{attribute 'linkalways'} 
{attribute 'no_explicit_call' := 'This FB is a CLASS and must be accessed using methods or properties'}
{attribute 'enable_dynamic_creation'}
FUNCTION_BLOCK _ETcVnColorMapSize EXTENDS EnumDatatypeBase
VAR
	localData : ETcVnColorMapSize;
	activeData : REFERENCE TO ETcVnColorMapSize;
	enumBaseDatatype : _UDINT(localData);
END_VAR

METHOD PRIVATE AddLocalEnumeration
VAR_INPUT
	Enumeration : T_MAXSTRING;
	Value : ETcVnColorMapSize;
END_VAR
AddEnumeration(Enumeration, Value);
END_METHOD

PROPERTY PUBLIC Address : PVOID
GET
Address := ADR(activeData);
END_GET
END_PROPERTY

METHOD PUBLIC ClearReference
VAR_INPUT
END_VAR
activeData REF= localData;
SetBaseDatatypeReference();
END_METHOD

METHOD PUBLIC Clone : I_Datatype
VAR
    pClone : POINTER TO _ETcVnColorMapSize;
END_VAR
pClone := __NEW(_ETcVnColorMapSize(InitialValue := Value));
Clone := pClone^;
END_METHOD

METHOD FB_init : BOOL
VAR_INPUT
	bInitRetains : BOOL; // if TRUE, the retain variables are initialized (warm start / cold start)
	bInCopyCode : BOOL;  // if TRUE, the instance afterwards gets moved into the copy code (online change)
	InitialValue : ETcVnColorMapSize;
END_VAR
localData := InitialValue;
AddBaseDatatype(enumBaseDatatype);
ClearReference();

AddLocalEnumeration('TCVN_CMS_256', ETcVnColorMapSize.TCVN_CMS_256);
AddLocalEnumeration('TCVN_CMS_65536', ETcVnColorMapSize.TCVN_CMS_65536);
END_METHOD

PROPERTY PUBLIC Identifier : T_MAXSTRING
GET
Identifier := 'ETcVnColorMapSize';
END_GET
END_PROPERTY

METHOD IsEnumeratorValueEqual : BOOL
VAR_INPUT
	Enumerator : I_KeyValueForwardEnumerator;
END_VAR
VAR
	storedValue : ETcVnColorMapSize;
END_VAR
IF NOT Enumerator.TryGet(storedValue) THEN
	RETURN;
END_IF

IsEnumeratorValueEqual := storedValue = activeData;
END_METHOD

METHOD PUBLIC MakeReferenceTo
VAR_INPUT
	ReferenceTarget : REFERENCE TO ETcVnColorMapSize;
END_VAR
activeData REF= ReferenceTarget;
SetBaseDatatypeReference();
END_METHOD

METHOD PROTECTED SetBaseDatatypeReference
VAR_INPUT
END_VAR
enumBaseDatatype.MakeReferenceTo(activeData);
END_METHOD

PROPERTY PUBLIC Size : UDINT
GET
Size := SIZEOF(activeData);
END_GET
END_PROPERTY

METHOD TryMakeReferenceTo : BOOL
VAR_INPUT
	Target : I_Datatype;
END_VAR
VAR
	targetAsEnum : I_EnumDatatype;
	pTargetData : POINTER TO ETcVnColorMapSize;
END_VAR
IF NOT Target.TryResolveAsEnumDatatype(targetAsEnum) THEN
	RETURN;
END_IF

IF targetAsEnum.Identifier <> Identifier THEN
	RETURN;
END_IF

pTargetData := Target.Address;
activeData REF= pTargetData^;
SetBaseDatatypeReference();
TryMakeReferenceTo := TRUE;
END_METHOD

PROPERTY PUBLIC Value : ETcVnColorMapSize
GET
Value := activeData;
END_GET
SET
activeData := Value;
END_SET
END_PROPERTY

END_FUNCTION_BLOCK

(* stored: Version 1.1.0.1, ProductVersion 3.1.4024.12
   POU _ETcVnColorMapSize: Id {3ff04702-16b4-09ab-01b0-cb3482cbb264}, SpecialFunc None
   Folder Constructor: Id {b8dfe9b5-ce15-023c-2ec2-92561a12cffe}
   Folder Private: Id {3649259b-32fa-072a-0861-9ae986f0a20c}
   Folder Protected: Id {7c534b05-1932-0159-3c33-ef5584caf8ae}
   Method AddLocalEnumeration: Id {cba97d69-b954-0b06-2654-beef1980051b}
   Property Address: Id {70222fa3-4b17-035a-0175-574d473a79f1}
   Get Get: Id {ac1edc10-2816-0f49-200c-b8edb701753e}
   Method ClearReference: Id {36299498-176e-00dc-3bde-8dd9fab5c4b5}
   Method Clone: Id {31486a7b-847d-0c8d-1164-cff563f2ffe6}
   Method FB_init: Id {473366ce-966d-0d59-3759-ebaf57c507b7}
   Property Identifier: Id {ab47df75-3f06-0989-0f44-e3eebad581e1}
   Get Get: Id {dabe0aba-0e4b-03bb-3d96-e8776ba66d9e}
   Method IsEnumeratorValueEqual: Id {b7525c9e-5b2c-0539-04d1-fb5a04646780}
   Method MakeReferenceTo: Id {5f9304f4-e89b-099a-0170-eb94090ff4ed}
   Method SetBaseDatatypeReference: Id {97880e42-0786-043e-3a26-4bb2294b6ec2}
   Property Size: Id {2f27e78f-73bf-0266-162e-32dbc09076fe}
   Get Get: Id {2789b148-75ce-0807-18b9-ca132a36810b}
   Method TryMakeReferenceTo: Id {89baca98-d467-0cb9-2ebc-290e7be37815}
   Property Value: Id {c2a3d649-3a64-05ad-3498-ca9963e7208d}
   Get Get: Id {92c23e03-0961-0a84-2c91-85f43000c4d8}
   Set Set: Id {c599ca1f-12bf-034b-3a5c-ad91f9277bb1} *)
